// TIA Portal V18 export
DATA_BLOCK "HSsDI"   // DB1025
{ S7_Optimized_Access := 'FALSE' }
VERSION : 0.1
// stored: AutoNumber false, DBAccessibleFromOPCUA true, IsOnlyStoredInLoadMemory false, IsWriteProtectedInAS false
   VAR
      Requests { S7_SetPoint := 'True'} : "UDT_HSsDI";
   END_VAR
BEGIN
END_DATA_BLOCK
